(* CODESYS project xd.project

Project tree, tasks and I/O mapping:
  Device : CODESYS Control Win V3, 3S - Smart Software Solutions GmbH, order no. 305021, version 3.5.7.20
    application Application
      libraries: Standard, * (System)
      task MainTask (cyclic, interval t#20ms, priority 1) calls PLC_PRG
      program PLC_PRG [LD]
      Symbols
*)

// Device/Application/PLC_PRG
PROGRAM PLC_PRG
VAR
	EB0:BYTE;
	AB0:BYTE;
	T1: TON;
	xd: TIME;
END_VAR

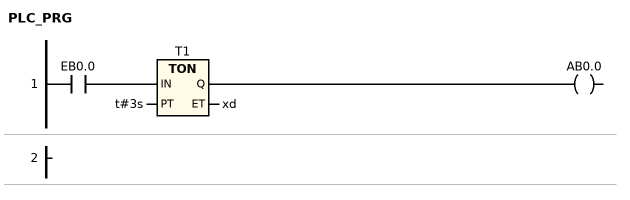
// NETWORK 1
T1(IN := EB0.0, PT := t#3s, ET => xd); // TON
AB0.0 := T1.Q;

// NETWORK 2

END_PROGRAM
